# EPICS autosave request: calcApp/Db/userArrayCalcs10more_settings.req
# FILE... userArrayCalcs10_settings.req
# USAGE.. userArrayCalcs10.db fields autosave'd.

file acalcout_settings.req P=$(P)userArrayCalc$(N1)
$(P)userStringSeq$(N1)Enable
file acalcout_settings.req P=$(P)userArrayCalc$(N2)
$(P)userStringSeq$(N2)Enable
file acalcout_settings.req P=$(P)userArrayCalc$(N3)
$(P)userStringSeq$(N3)Enable
file acalcout_settings.req P=$(P)userArrayCalc$(N4)
$(P)userStringSeq$(N4)Enable
file acalcout_settings.req P=$(P)userArrayCalc$(N5)
$(P)userStringSeq$(N5)Enable
file acalcout_settings.req P=$(P)userArrayCalc$(N6)
$(P)userStringSeq$(N6)Enable
file acalcout_settings.req P=$(P)userArrayCalc$(N7)
$(P)userStringSeq$(N7)Enable
file acalcout_settings.req P=$(P)userArrayCalc$(N8)
$(P)userStringSeq$(N8)Enable
file acalcout_settings.req P=$(P)userArrayCalc$(N9)
$(P)userStringSeq$(N9)Enable
file acalcout_settings.req P=$(P)userArrayCalc$(N10)
$(P)userStringSeq$(N10)Enable
